(* CoDeSys 2.3 export: PLCSUPLIB.EXP *)
(* Libraries: E:\Projekte\WebSocketLib\WebSocket.lib 7.1.13 10:17:33, Ethernet.lib 2.12.10 13:48:32, IecSfc.lib 13.4.06 15:51:28, Standard.lib 2.12.10 13:48:34, SYSLIBCALLBACK.LIB 2.12.10 13:48:32, SysLibSockets.lib 10.2.11 08:20:54, SysLibStr.lib 2.12.10 13:48:34, SysLibTime.lib 2.12.10 13:48:32, SysTaskInfo.lib 2.12.10 13:48:32, WagoLibBase64_01.lib 19.9.11 07:14:42, WagoLibEthernet_01.lib 20.2.12 16:40:34, WagoLibSHA1.lib 19.9.11 07:14:42 *)

(* Global variable list: Globale_Konstanten *)
VAR_GLOBAL CONSTANT
	MAX_SUBSCRIPTIONS		:	BYTE := 100;
END_VAR

(* Data type *)
TYPE Address :
STRUCT
	bitCount	:	BYTE;
	offset		:	UINT;
END_STRUCT
END_TYPE

(* Data type *)
TYPE Subscription :
STRUCT

	address		:	Address;

	active			:	BOOL := FALSE;

	oldValue		:	DWORD;
END_STRUCT
END_TYPE

(* POU PLC_PRG, ST *)
PROGRAM PLC_PRG
VAR
	wsSubscriber				:	wsSubscriber;
	WebSocket				:	WebSocket;
	tcpServer					:	TCP_Server;

	vBoolOne AT %MX0.0		:	BOOL;
	vBoolTwo AT %MX0.1		:	BOOL;
	vBoolThree AT %MX0.2	:	BOOL;
	vByteOne AT %MB2		:	BYTE;
	vWordOne AT %MW3		:	WORD;
	vDWordOne AT %MD6	:	DWORD;
END_VAR
(*invoke the wsSubscriber module simply like this and make this programm a
   free running task *)
wsSubscriber(WebSocket := ADR(WebSocket), tcpServer := ADR(tcpServer));
END_PROGRAM

(* POU wsSubscriber, ST *)
FUNCTION_BLOCK wsSubscriber
VAR_INPUT
	WebSocket		:	POINTER TO WebSocket;
	tcpServer			:	POINTER TO TCP_Server;
END_VAR
VAR_OUTPUT
END_VAR
VAR CONSTANT
	WRITE						:	BYTE := 0;
	READ						:	BYTE := 1;
	SUBSCRIBE				:	BYTE := 2;
	UNSUBSCRIBE			:	BYTE := 3;
END_VAR
VAR

	rcvPkt				:	Packet;
	sendPkt			:	Packet;

	subs				:	ARRAY[0..MAX_SUBSCRIPTIONS] OF Subscription;

	functionCode		:	BYTE;

	address			:	Address;

	vBoolValue		:	BOOL;
	pByte				:	POINTER TO BYTE;

	I, J					:	BYTE;

	numberOfSubs	:	INT := 0;

	oldState			:	BYTE := 0;

END_VAR
WebSocket^(tcpServer := tcpServer, rcvPkt := rcvPkt, sendPkt := sendPkt);

(*  in case information are available on the websocket port *)
IF (rcvPkt.size > 0 AND WebSocket^.state = WebSocket^.OPEN) THEN

	(* get the function code of the request *)
	functionCode := getFunctionCode(ADR(rcvPkt));

	(* handle read request *)
	IF (functionCode = READ) THEN

		address:= getAddress(ADR(rcvPkt), 0);
		sendReadAnswer(ADR(sendPkt), address);

	(* handle write request *)
	ELSIF (functionCode = WRITE) THEN

		address := getAddress(ADR(rcvPkt), 0);
		setValue(ADR(rcvPkt), address);
		sendWriteAnswer(ADR(sendPkt), address);

	(* handle subscribe request *)
	ELSIF (functionCode = subscribe) THEN

		(* read subscriptions till zero bitcount arrives *)
		numberOfSubs := subscribe(ADR(rcvPkt), ADR(subs));

		IF (numberOfSubs = MAX_SUBSCRIPTIONS) THEN
			sendOutOfSubsAnswer(ADR(sendPkt));
		ELSE
			sendSubscribeAnswer(ADR(sendPkt), numberOfSubs);
		END_IF

	(* handle unsubscribe request (not implemented yet) *)
	ELSIF (functionCode = unsubscribe) THEN

		(* read subscriptions till zero bitcount arrives *)
		unsubscribe(ADR(rcvPkt), ADR(subs));

	END_IF

	(* free received bytes *)
	rcvPkt.size := 0;

END_IF

(* in case no other packet should be send or not sending process is ongoing check
    the subscriptions and send updates *)
IF (sendPkt.size = 0 AND WebSocket^.state = WebSocket^.OPEN AND NOT WebSocket^.sending) THEN
	FOR I:= 0 TO MAX_SUBSCRIPTIONS DO

		IF (subs[I].active) THEN
			sendUpdate(ADR(sendPKt), ADR(subs[I]));
		END_IF

	END_FOR

END_IF

(* if the websocket connection is closed then remove all subscriptions *)
IF (oldState = WebSocket^.OPEN AND WebSocket^.state = WebSocket^.CLOSED) THEN
	FOR I:= 0 TO MAX_SUBSCRIPTIONS DO

		subs[I].active := FALSE;

	END_FOR

END_IF

oldState := WebSocket^.state;
END_FUNCTION_BLOCK

(* POU private/subscribe, ST *)
FUNCTION subscribe : INT
VAR_INPUT
	rcvPkt		:	POINTER TO Packet;
	subs		:	POINTER TO ARRAY[0..MAX_SUBSCRIPTIONS] OF Subscription;
END_VAR
VAR
	I, J			:	BYTE;
	address	:	Address;

END_VAR
subscribe := 0;

I := 0; J := 0;
address := getAddress(rcvPkt, 0);
WHILE (address.bitCount > 0 AND i < 122) DO

	WHILE (subs^[J].active AND J < MAX_SUBSCRIPTIONS) DO
		J := J + 1;
		subscribe := subscribe + 1;
	END_WHILE;

	IF (subscribe = MAX_SUBSCRIPTIONS) THEN
		RETURN;
	END_IF

	subs^[J].active := TRUE;

	subs^[j].address := address;

	I := I + 3;

	address := getAddress(rcvPkt, I);
END_WHILE

WHILE (J < MAX_SUBSCRIPTIONS) DO
	IF (subs^[j].active) THEN
		subscribe := subscribe + 1;
	END_IF
	J := J + 1;
END_WHILE;
END_FUNCTION

(* POU private/getAddress, ST *)
FUNCTION getAddress : Address
VAR_INPUT
	rcvPacket		:	POINTER TO Packet;
	offset			:	BYTE := 0;
END_VAR
VAR
	address		:	POINTER TO INT;
END_VAR
getAddress.bitCount := getBitCount(rcvPacket, offset);
getAddress.offset := SHL(rcvPacket^.data[offset + 1], 8) + rcvPacket^.data[offset+2];
END_FUNCTION

(* POU private/getBitCount, ST *)
FUNCTION getBitCount : BYTE
VAR_INPUT
	rcvPacket		:	POINTER TO Packet;
	offset			:	BYTE := 0;
END_VAR
VAR
END_VAR
IF (rcvPacket^.data[offset].7) THEN
	getBitCount := 1;
	RETURN;
ELSIF (rcvPacket^.data[offset].6) THEN
	getBitCount := 8;
	RETURN;
ELSIF (rcvPacket^.data[offset].5) THEN
	getBitCount := 16;
	RETURN;
ELSIF (rcvPacket^.data[offset].4) THEN
	getBitCount := 32;
	RETURN;
ELSIF (rcvPacket^.data[offset].3) THEN
	getBitCount := 64;
ELSE
	getBitCount := 0;
END_IF
END_FUNCTION

(* POU private/unsubscribe, ST *)
FUNCTION unsubscribe : BOOL
VAR_INPUT
	rcvPkt		:	POINTER TO Packet;
	subs		:	POINTER TO ARRAY[0..MAX_SUBSCRIPTIONS] OF Subscription;
END_VAR
VAR
	I, J			:	BYTE;
	address	:	Address;
END_VAR
I := 0; J := 0;
address := getAddress(rcvPkt, 0);
WHILE (address.bitCount > 0 AND I < 122) DO

	WHILE (subs^[J].active) DO
		J := (J + 1) MOD MAX_SUBSCRIPTIONS;
	END_WHILE;

	subs^[J].active := FALSE;

	I := I + 3;

	address := getAddress(rcvPkt, I);

END_WHILE
END_FUNCTION

(* POU private/getFunctionCode, ST *)
FUNCTION getFunctionCode : BYTE
VAR_INPUT
	rcvPacket		:	POINTER TO Packet;
END_VAR
VAR
END_VAR
getFunctionCode.0 := rcvPacket^.data[0].0;
getFunctionCode.1 := rcvPacket^.data[0].1;
END_FUNCTION

(* POU messages/sendReadAnswer, ST *)
FUNCTION sendReadAnswer : BOOL
VAR_INPUT

	sendPkt		:	POINTER TO Packet;
	address		:	Address;

END_VAR
VAR

	value				:	DWORD;

END_VAR
sendPkt^.data[0] := 0;
sendPkt^.data[0].0 := 1;
sendPKt^.data[0].2 := 1;
sendPkt^.data[1] := UINT_TO_BYTE(SHR(address.offset, 8));
sendPkt^.data[2] := UINT_TO_BYTE(SHR(SHL(address.offset, 8), 8));

IF (address.bitCount = 1) THEN
	IF (getBitValue(address)) THEN
		sendPkt^.data[3] := 255;
	ELSE
		sendPkt^.data[3] := 0;
	END_IF

	sendPkt^.data[0].7 := TRUE;

	sendPkt^.size := sendPkt^.size + 4;

ELSIF (address.bitCount = 8) THEN

	sendPkt^.data[0].6 := TRUE;

	sendPkt^.data[3] := getByteValue(address);

	sendPkt^.size := sendPkt^.size + 4;

ELSIF (address.bitCount = 16) THEN

	sendPkt^.data[0].5 := TRUE;

	value := getWordValue(address);

	sendPkt^.data[3] := DWORD_TO_BYTE(SHR(value, 8));
	sendPkt^.data[4] := DWORD_TO_BYTE(SHR(SHL(value, 8), 8));

	sendPkt^.size := sendPkt^.size + 5;

ELSIF (address.bitCount = 32) THEN

	sendPkt^.data[0].4 := TRUE;

	value := getDWordValue(address);

	sendPkt^.data[3] := DWORD_TO_BYTE(SHR(value, 24));
	sendPkt^.data[4] := DWORD_TO_BYTE(SHR(SHL(value, 8), 24));
	sendPkt^.data[5] := DWORD_TO_BYTE(SHR(SHL(value, 16), 24));
	sendPkt^.data[6] := DWORD_TO_BYTE(SHR(SHL(value, 24), 24));

	sendPkt^.size := sendPkt^.size + 7;

END_IF
END_FUNCTION

(* POU values/getBitValue, ST *)
FUNCTION getBitValue : BOOL
VAR_INPUT
	address		:	Address;
END_VAR
VAR
	offset			:	UINT;
	modulo		: 	BYTE;
	pByte			:	POINTER TO BYTE;
END_VAR
modulo := INT_TO_BYTE(address.offset MOD 8);
offset := TRUNC((address.offset - modulo) / 8 );

pByte := ADR(%MB0) + offset;

getBitValue := getBit(pByte^, modulo);
END_FUNCTION

(* POU private/getBit, ST *)
FUNCTION getBit : BOOL
VAR_INPUT
	src		: 		BYTE;
	index	:		BYTE;
END_VAR
VAR
END_VAR
IF (index = 0) THEN
	getBit:= src.0;
ELSIF (index = 1) THEN
	getBit := src.1;
ELSIF (index = 2) THEN
	getBit := src.2;
ELSIF (index = 3) THEN
	getBit := src.3;
ELSIF (index = 4) THEN
	getBit := src.4;
ELSIF (index = 5) THEN
	getBit := src.5;
ELSIF (index = 6) THEN
	getBit := src.6;
ELSIF (index = 7) THEN
	getBit := src.7;
END_IF
END_FUNCTION

(* POU values/getByteValue, ST *)
FUNCTION getByteValue : BYTE
VAR_INPUT
	address		:	Address;
END_VAR
VAR
	pByte			:	POINTER TO BYTE;
END_VAR
pByte := ADR(%MB0) + address.offset;
getByteValue := pByte^;
END_FUNCTION

(* POU values/getWordValue, ST *)
FUNCTION getWordValue : WORD
VAR_INPUT
	address		:	Address;
END_VAR
VAR
	pWord			:	POINTER TO WORD;
END_VAR
pWord := ADR(%MW0) + address.offset;
getWordValue := pWord^;
END_FUNCTION

(* POU values/getDWordValue, ST *)
FUNCTION getDWordValue : DWORD
VAR_INPUT
	address		:	Address;
END_VAR
VAR
	pdWord		:	POINTER TO DWORD;
END_VAR
pdWord := ADR(%MD0) + address.offset;
getDWordValue := pdWord^;
END_FUNCTION

(* POU private/setValue, ST *)
FUNCTION setValue : BOOL
VAR_INPUT
	rcvPkt			:	POINTER TO Packet;
	address		:	Address;
END_VAR
VAR
END_VAR
IF (address.bitCount = 1) THEN
	IF (rcvPkt^.data[3] = 255) THEN
		setBitValue(address, TRUE);
	ELSIF (rcvPkt^.data[3] = 0) THEN
		setBitValue(address, FALSE);
	END_IF
ELSIF (address.bitCount = 8) THEN
	setByteValue(address, rcvPkt^.data[3]);
ELSIF (address.bitCount = 16) THEN
	setWordValue(address, SHL(rcvPkt^.data[3], 8) + rcvPkt^.data[4]);
ELSIF (address.bitCount = 32) THEN
	setDWordValue(address, SHL(rcvPkt^.data[3], 24) + SHL(rcvPkt^.data[4], 16) + SHL(rcvPkt^.data[5], 8) + rcvPkt^.data[6]);
END_IF
END_FUNCTION

(* POU values/setBitValue, ST *)
FUNCTION setBitValue : BOOL
VAR_INPUT
	address		:	Address;
	value			:	BOOL;
END_VAR
VAR
	offset			:	UINT;
	modulo		:	BYTE;
	pByte			:	POINTER TO BYTE;
END_VAR
modulo := INT_TO_BYTE(address.offset MOD 8);
offset := TRUNC((address.offset - modulo) / 8 );
pByte := ADR(%MB0) + offset;
pByte^ := setBit(pByte^, modulo, value);
END_FUNCTION

(* POU private/setBit, ST *)
FUNCTION setBit : BYTE
VAR_INPUT
	src			:	BYTE;
	index		:	BYTE;
	value		:	BOOL;
END_VAR
VAR
END_VAR
setBit := src;
IF (index = 0) THEN
	setBit.0:= value;
ELSIF (index = 1) THEN
	setBit.1 := value;
ELSIF (index = 2) THEN
	setBit.2 := value;
ELSIF (index = 3) THEN
	setBit.3 := value;
ELSIF (index = 4) THEN
	setBit.4 := value;
ELSIF (index = 5) THEN
	setBit.5 := value;
ELSIF (index = 6) THEN
	setBit.6 := value;
ELSIF (index = 7) THEN
	setBit.7 := value;
END_IF
END_FUNCTION

(* POU values/setByteValue, ST *)
FUNCTION setByteValue : BOOL
VAR_INPUT
	address		:	Address;
	value			:	BYTE;
END_VAR
VAR
	pByte			:	POINTER TO BYTE;
END_VAR
pByte := ADR(%MB0) + address.offset;
pByte^ := value;
END_FUNCTION

(* POU values/setWordValue, ST *)
FUNCTION setWordValue : BOOL
VAR_INPUT
	address		:	Address;
	value			:	WORD;
END_VAR
VAR
	pWord			:	POINTER TO WORD;
END_VAR
pWord := ADR(%MW0) + address.offset;
pWord^ := value;
END_FUNCTION

(* POU values/setDWordValue, ST *)
FUNCTION setDWordValue : BOOL
VAR_INPUT
	address		:	Address;
	value			:	DWORD;
END_VAR
VAR
	pDWord		:	POINTER TO DWORD;
END_VAR
pDWord := ADR(%MD0) + address.offset;
pDWord^ := value;
END_FUNCTION

(* POU messages/sendWriteAnswer, ST *)
FUNCTION sendWriteAnswer : BOOL
VAR_INPUT

	sendPkt		:	POINTER TO Packet;
	address		:	Address;
END_VAR
VAR
END_VAR
sendPkt^.data[0] := 0;
sendPkt^.data[0].2 := 1;
sendPkt^.data[1] := INT_TO_BYTE(SHR(address.offset, 8));
sendPkt^.data[2] := INT_TO_BYTE(SHR(SHL(address.offset, 8), 8));

sendPkt^.size := 3;
END_FUNCTION

(* POU messages/sendOutOfSubsAnswer, ST *)
FUNCTION sendOutOfSubsAnswer : BOOL
VAR_INPUT
	sendPkt	:	POINTER TO Packet;
END_VAR
VAR
END_VAR
sendPkt^.data[0] := 2 + 8;
sendPkt^.data[1] := 2;
END_FUNCTION

(* POU messages/sendSubscribeAnswer, ST *)
FUNCTION sendSubscribeAnswer : BOOL
VAR_INPUT
	sendPkt			:	POINTER TO Packet;
	numberOfSubs	:	UINT;
END_VAR
VAR
END_VAR
sendPkt^.data[0] := 6;
sendPkt^.data[1] := UINT_TO_BYTE(SHR(numberOfSubs, 8));
sendPkt^.data[2] := UINT_TO_BYTE(SHR(SHL(numberOfSubs, 8), 8));
sendPkt^.size := 3;
END_FUNCTION

(* POU messages/sendUpdate, ST *)
FUNCTION sendUpdate : BOOL
VAR_INPUT

	sendPkt		:	POINTER TO Packet;
	pSub			:	POINTER TO Subscription;

END_VAR
VAR

	offset				:	UINT;

	address			:	Address;

	value				:	DWORD;

END_VAR
offset := sendPkt^.size;
sendPKt^.data[offset] := 2 + 12;

address := pSub^.address;

sendPkt^.data[offset + 1] := INT_TO_BYTE(SHR(address.offset, 8));
sendPkt^.data[offset + 2] := INT_TO_BYTE(SHR(SHL(address.offset, 8), 8));

IF (address.bitCount = 1) THEN
	IF (getBitValue(address)) THEN
		value := 255;
	ELSE
		value := 0;
	END_IF

	IF (value <> pSub^.oldValue) THEN
		sendPkt^.data[offset].7 := TRUE;
		sendPkt^.data[offset + 3] := DWORD_TO_BYTE(value);
		sendPkt^.size := sendPkt^.size + 4;
		pSub^.oldValue := value;
	END_IF


ELSIF (address.bitCount = 8) THEN

	value := getByteValue(address);

	IF (value <> pSub^.oldValue) THEN
		sendPkt^.data[offset].6 := TRUE;
		sendPkt^.data[offset + 3] := DWORD_TO_BYTE(value);
		sendPkt^.size := sendPkt^.size + 4;

		pSub^.oldValue := value;

	END_IF

ELSIF (address.bitCount = 16) THEN

	value := getWordValue(address);

	IF (value <> pSub^.oldValue) THEN
		sendPkt^.data[offset].5 := TRUE;

		sendPkt^.data[offset + 3] := DWORD_TO_BYTE(SHR(value, 8));
		sendPkt^.data[offset + 4] := DWORD_TO_BYTE(SHR(SHL(value, 8), 8));

		sendPkt^.size := sendPkt^.size + 5;

		pSub^.oldValue := value;
	END_IF

ELSIF (address.bitCount = 32) THEN

	value := getDWordValue(address);

	IF (value <> pSub^.oldValue) THEN
		sendPkt^.data[offset].4 := TRUE;

		sendPkt^.data[offset + 3] := DWORD_TO_BYTE(SHR(value, 24));
		sendPkt^.data[offset + 4] := DWORD_TO_BYTE(SHR(SHL(value, 8), 24));
		sendPkt^.data[offset + 5] := DWORD_TO_BYTE(SHR(SHL(value, 16), 24));
		sendPkt^.data[offset + 6] := DWORD_TO_BYTE(SHR(SHL(value, 24), 24));

		sendPkt^.size := sendPkt^.size + 7;

		pSub^.oldValue := value;

	END_IF

END_IF
END_FUNCTION
